// TIA Portal V16 export
// export: Created 2024-05-10T06:46:45.1534973Z, ExportSetting WithDefaults, DisplayName Totally Integrated Automation Portal, DisplayVersion V16, DisplayName TIA Portal Version Control Interface, DisplayVersion V16, DisplayName TIA Portal Openness, DisplayVersion V16, DisplayName STEP 7 Professional, DisplayVersion V16, DisplayName STEP 7 Safety, DisplayVersion V16, DisplayName WinCC Professional, DisplayVersion V16
VAR_GLOBAL   // PLC tag table "104输出点变量表"
   EN_INV1正转 AT %Q2.0 : Bool;
   EN_INV1反转 AT %Q2.1 : Bool;
   EN_INV1速度 AT %Q2.2 : Bool;
   EN_INV1复位 AT %Q2.3 : Bool;
   EN_阻挡下降 AT %Q2.5 : Bool;
   EN_提升机上升 AT %Q2.6 : Bool;
   EN_提升机下降 AT %Q2.7 : Bool;
   EX_INV2正转 AT %Q3.0 : Bool;
   EX_INV2反转 AT %Q3.1 : Bool;
   EX_INV2速度 AT %Q3.2 : Bool;
   EX_INV2复位 AT %Q3.3 : Bool;
   EX_阻挡下降 AT %Q3.5 : Bool;
   EX_提升机上升 AT %Q3.6 : Bool;
   EX_提升机下降 AT %Q3.7 : Bool;
   ST01上阻挡下降 AT %Q4.1 : Bool;
   ST01下阻挡下降 AT %Q4.3 : Bool;
   ST02上阻挡下降 AT %Q4.5 : Bool;
   ST02下阻挡下降 AT %Q4.7 : Bool;
   ST03上阻挡下降 AT %Q5.1 : Bool;
   ST03下阻挡下降 AT %Q5.3 : Bool;
   ST04上阻挡下降 AT %Q5.5 : Bool;
   ST05上阻挡下降 AT %Q5.7 : Bool;
   前段_INV3正转 AT %Q8.0 : Bool;
   前段_INV3速度1 AT %Q8.1 : Bool;
   前段_INV3速度2 AT %Q8.2 : Bool;
   前段_INV3复位 AT %Q8.3 : Bool;
   前段_INV4正转 AT %Q8.4 : Bool;
   前段_INV4速度1 AT %Q8.5 : Bool;
   前段_INV4速度2 AT %Q8.6 : Bool;
   前段_INV4复位 AT %Q8.7 : Bool;
   后段_INV5正转 AT %Q9.0 : Bool;
   后段_INV5速度1 AT %Q9.1 : Bool;
   后段_INV5速度2 AT %Q9.2 : Bool;
   后段_INV5复位 AT %Q9.3 : Bool;
   后段_INV6正转 AT %Q9.4 : Bool;
   后段_INV6速度1 AT %Q9.5 : Bool;
   后段_INV6速度2 AT %Q9.6 : Bool;
   后段_INV6复位 AT %Q9.7 : Bool;
   ST06上阻挡下降 AT %Q10.1 : Bool;
   ST07上阻挡下降 AT %Q10.3 : Bool;
   ST08上阻挡下降 AT %Q10.5 : Bool;
   ST09上阻挡下降 AT %Q11.1 : Bool;
   ST10上阻挡下降 AT %Q11.3 : Bool;
   ST11上阻挡下降 AT %Q11.5 : Bool;
   ST12上阻挡下降 AT %Q11.7 : Bool;
   ST01放行LED AT %Q12.0 : Bool;
   ST02放行LED AT %Q12.1 : Bool;
   ST03放行LED AT %Q12.2 : Bool;
   ST04放行LED AT %Q12.3 : Bool;
   ST05放行LED AT %Q12.4 : Bool;
   ST06放行LED AT %Q12.5 : Bool;
   ST07放行LED AT %Q13.0 : Bool;
   ST08放行LED AT %Q13.1 : Bool;
   ST09放行LED AT %Q13.2 : Bool;
   ST10放行LED AT %Q13.3 : Bool;
   ST11放行LED AT %Q13.4 : Bool;
   ST12放行LED AT %Q13.5 : Bool;
END_VAR
